FUNCTION_BLOCK FB_HVAC_RND_ModbusApadtor EXTENDS FB_BaseDevice

VAR
	
	// ----------------- Modbus Variables -----------//
	// Written in accordance with the modbus manuial supplied by vendor
	// https://drive.google.com/file/d/1Gl1Z8UXsnYqQFCh63b19Rq_Jpmyq9qef/view?usp=sharing
	
	// -------------------READ ONLY ---------------//
	bReady: BOOL;
	
	// -------------------READ / WRITE ---------------//
	bManagedDIINetAdr: BOOL;
	bDIINetMasterFlag: BOOL;
	bDIINet_Comms_StartStopFlag: BOOL;
	
	
	
END_VAR

END_FUNCTION_BLOCK

(* stored: Version 1.1.0.1, ProductVersion 3.1.4024.12
   POU FB_HVAC_RND_ModbusApadtor: Id {04beb52c-ae32-40c4-bc43-713399989349}, SpecialFunc None *)
